PROGRAM MAIN
VAR
	//if true dan rijdt hij autonoom
	Autonoom : BOOL;	
	
	//voor inleen pedal
	InputNum AT%I* : INT;
	Percentage : REAL;

	//Voor Motion
	fbReadXaxisStatus: MC_ReadStatus;	
END_VAR

IF Autonoom THEN
	Percentage := Scaling(Input:= InputNum, Imin:= 0, Imax:= 32767, Qmin:= 0, Qmax:= 100);
END_IF

fbReadXaxisStatus(
	Axis:=GVL_NC.stXAxis , 
	Enable:= GVL_AxisCtr.bXAxisEnable , 
	Valid=> , Busy=> , Error=> , 
	ErrorID=> , ErrorStop=> , 
	Disabled=> , Stopping=> , 
	StandStill=> , DiscreteMotion=> , 
	ContinuousMotion=> , SynchronizedMotion=> , 
	Homing=> , ConstantVelocity=> , 
	Accelerating=> , Decelerating=> , 
	Status=> GVL_NC.stXaxisStatus);
	POUNCPowerOn();
	movements();

END_PROGRAM

(* stored: Version 1.1.0.1, ProductVersion 3.1.4024.3
   POU MAIN: Id {f48db1e3-9dde-48d5-bccc-d0cb3279a1dc}, SpecialFunc None *)
